// TwinCAT 3 PLC project Untitled1
// ProgramVersion: 3.1.4023.0
// libraries:
//   Tc2_ControllerToolbox, * (Beckhoff Automation GmbH)
//   Tc2_Standard, * (Beckhoff Automation GmbH)
//   Tc2_System, * (Beckhoff Automation GmbH)
//   Tc3_EventLogger, * (Beckhoff Automation GmbH)
//   Tc3_Module, * (Beckhoff Automation GmbH)
//   VisuDialogs, * (System)
//   VisuSymbols,3.5.10.0,System
// project tree:
//   DUTs/ AlarmState.TcDUT
//   / GlobalTextList.TcGTLO, PlcTask.TcTTO, Visualization Manager.TcVMO (not stored)
//   GVLs/ gAL.TcGVL
//   POUs/ ControlSystem.TcPOU, FB_EmergencySystem.TcPOU, FB_defaultValues.TcPOU, MAIN.TcPOU, FB_Tank1HysteresisBuffer.TcPOU
// real-time tasks:
//   TASK PlcTask: cycle T#10ms, priority 20, ADS port 350
// I/O:
//   DEVICE Device 1 (EtherCAT), AmsNetId 5.112.67.239.2.1
//     Term 7 (EK1200) [EK1200-5000 EtherCAT Power supply (2A E-Bus)]
//       Term 2 (EL4004) [EL4004 4Ch. Ana. Output 0-10V, 12bit]
//       Term 3 (EL4004) [EL4004 4Ch. Ana. Output 0-10V, 12bit]
//       Term 8 (EL3024) [EL3024 4Ch. Ana. Input 4-20mA DIFF]
//       Term 9 (EL3024) [EL3024 4Ch. Ana. Input 4-20mA DIFF]
//       Term 12 (EL1859) [EL1859 8Ch. Dig. Input 24V, 3ms, 8Ch. Dig. Output 24V, 0.5A]
//       Term 13 (EL9011) [EL9011 End Terminal]
// variable links:
//   Untitled1/Untitled1 Instance <-> Device 1 (EtherCAT)/Term 7 (EK1200)/Term 12 (EL1859)
//     PlcTask Inputs/MAIN.EMERGENCY_STOP <-> Channel 1/EMERGENCY STOP
//     PlcTask Inputs/MAIN.Reset_Button <-> Channel 3/Reset Button
//     PlcTask Inputs/MAIN.Toggle_Button <-> Channel 2/Toggle Button
//     PlcTask Outputs/MAIN.Motor_Direction <-> Channel 10/Motor Direction
//     PlcTask Outputs/MAIN.Motor_ON_OFF <-> Channel 9/Motor ON/OFF
//   Untitled1/Untitled1 Instance <-> Device 1 (EtherCAT)/Term 7 (EK1200)/Term 2 (EL4004)
//     PlcTask Outputs/MAIN.Flow_Valve_1 <-> AO Outputs Channel 4/Flow_Valve_1
//     PlcTask Outputs/MAIN.Level_Valve_1 <-> AO Outputs Channel 1/Level_Valve_1
//     PlcTask Outputs/MAIN.Level_Valve_2 <-> AO Outputs Channel 2/Level_Valve_2
//     PlcTask Outputs/MAIN.Level_Valve_3 <-> AO Outputs Channel 3/Level_Valve_3
//   Untitled1/Untitled1 Instance <-> Device 1 (EtherCAT)/Term 7 (EK1200)/Term 3 (EL4004)
//     PlcTask Outputs/MAIN.Gas_Valve <-> AO Outputs Channel 1/Gas_Valve
//     PlcTask Outputs/MAIN.Mixer_Valve <-> AO Outputs Channel 2/Mixer_Valve
//     PlcTask Outputs/MAIN.Motor_speed <-> AO Outputs Channel 3/Motor_Speed
//   Untitled1/Untitled1 Instance <-> Device 1 (EtherCAT)/Term 7 (EK1200)/Term 8 (EL3024)
//     PlcTask Inputs/MAIN.Pressure_Differencial_Transmitter_1 <-> AI Standard Channel 1/PDT 1
//     PlcTask Inputs/MAIN.Pressure_Differencial_Transmitter_2 <-> AI Standard Channel 3/PDT 2
//     PlcTask Inputs/MAIN.Pressure_Transmitter_1 <-> AI Standard Channel 2/PT 1
//     PlcTask Inputs/MAIN.Pressure_Transmitter_3 <-> AI Standard Channel 4/PT 3
//   Untitled1/Untitled1 Instance <-> Device 1 (EtherCAT)/Term 7 (EK1200)/Term 9 (EL3024)
//     PlcTask Inputs/MAIN.Level_Transmitter_1 <-> AI Standard Channel 2/ Level Transmitter 1
//     PlcTask Inputs/MAIN.Level_Transmitter_2 <-> AI Standard Channel 3/Level Transmitter 2
//     PlcTask Inputs/MAIN.Pressure_Transmitter_2 <-> AI Standard Channel 1/PT 2
//     PlcTask Inputs/MAIN.Temperature_Transmitter <-> AI Standard Channel 4/Temperature Transmitter

CONFIGURATION Untitled1
    RESOURCE PLC ON TwinCAT3
        TASK PlcTask(INTERVAL := T#10ms, PRIORITY := 20);
        PROGRAM MAIN WITH PlcTask : MAIN;
        PROGRAM ControlSystem WITH PlcTask : ControlSystem;
        PROGRAM BufferTankFiller WITH PlcTask : BufferTankFiller;
    END_RESOURCE
END_CONFIGURATION

// ---- DUTs/AlarmState.TcDUT
{attribute 'qualified_only'}
{attribute 'strict'}
TYPE AlarmState :
	(
		AlarmActive := 0,
		AlarmClearPreTimer := 1,
		AlarmCleared := 2
	)USINT;
END_TYPE

// ---- GVLs/gAL.TcGVL
{attribute 'qualified_only'}
VAR_GLOBAL
	fbAlarm : FB_TcAlarm;	// Creates instance of integrated Alarm FB
	
	Motor_ON_OFF 	AT %Q* : BOOL := FALSE;	// Motor switch	
	// User Input as percentage, Declaration
	Flow_Valve_1_Percentage	: INT;	// Start values
	Level_Valve_1_Percentage: INT;	// From Manual
	Level_Valve_2_Percentage: INT;
	Level_Valve_3_Percentage: INT;
	Motor_speed_Percentage	: INT; // Start speed, ideal: 30-35%
END_VAR

// ---- POUs/MAIN.TcPOU
PROGRAM MAIN
VAR
	// ------ Linking variables to IO cards ------
		// --------- Outputs ---------
	Flow_Valve_1 	AT %Q* : INT;
	Level_Valve_1 	AT %Q* : INT;
	Level_Valve_2 	AT %Q* : INT;
	Level_Valve_3 	AT %Q* : INT;
	Gas_Valve 		AT %Q* : INT;
	Mixer_Valve 	AT %Q* : INT;
	Motor_speed 	AT %Q* : INT;	
	Motor_Direction AT %Q* : BOOL; 			// Don't touch
		// --------- Inputs ---------
			// Buttons
	Toggle_Button 	AT %I* :BOOL;	// Normally Open  (OFF), Green
	Reset_Button 	AT %I* : BOOL; 	// Normally Closed (ON), Red
	EMERGENCY_STOP 	AT %I* : BOOL; 	// Normally Closed (ON), Emergency Switch
			// Sensors
	Level_Transmitter_1 	AT %I* :INT;
	Level_Transmitter_2 	AT %I* :INT;
	Temperature_Transmitter AT %I* :INT;
	Pressure_Differencial_Transmitter_1 AT %I* : INT;
	Pressure_Differencial_Transmitter_2 AT %I* : INT;
	Pressure_Transmitter_1 AT %I* : INT ;
	Pressure_Transmitter_2 AT %I* : INT ;
	Pressure_Transmitter_3 AT %I* : INT ; 
	// ------ Linking variables to IO cards ------
	
	// ------- Display Input Variables ---------
		// Percentages
	LT1percent  : INT;
	LT2percent  : INT;
	TT1percent  : INT;
	PDT1percent : INT;
	PDT2percent : INT;
	PT1percent  : INT;
	PT2percent  : INT;
	PT3percent  : INT;
		// Actual values
	LT1mm 	: REAL;
	LT2mm 	: REAL;
	TT1c 	: REAL;
	PDT1bar : REAL;
	PDT2bar : REAL;
	PT1bar  : REAL;
	PT2bar  : REAL;
	PT3bar  : REAL;
		// Scaling variables
	bitMax 		: REAL := 32767;			// [bits]
	minPT 		: REAL := 0.06;				// [bar]
	maxPT 		: REAL := 6;				// [bar]
	deltaPT 	: REAL := maxPT - minPT;	// [bar]
	minPDT		: REAL := 0.004;			// [bar]
	maxPDT		: REAL := 0.4;				// [bar]
	deltaPDT	: REAL := maxPDT - minPDT;	// [bar]
	
	//maxLT 		: REAL := 304.8;			// [mm]
	minLT1  	: REAL := 37.0;				// [mm]
	minLT1bit  	: REAL := 270.0;			// [mm]
	minLT2  	: REAL := 42.0;				// [mm]
	kLT1		: REAL := 9.0/1694.0;		// [deltaMMmeasured/deltaBitmeasured]
	kLT2		: REAL := 9.0/1529.0;		// [deltaMMmeasured/deltaBitmeasured
	
	maxTT		: REAL := 250;				// [celsius]
	minTT		: REAL := -50;				// [celsius]
	deltaTT 	: REAL := maxTT - minTT;	// [celsius]
	// ------- Display Input Variables --------- 
	
	
		// Toggle Motor Statee with green button
	risingEdge : R_TRIG;
	elapsedDebounce : TIME;
	toggleMotor : BOOL;
	
	// ------------------ HMI ------------------
	Motor_ON : BOOL; 				// For HMI button
	ON_OFF 	 : STRING(10) := 'OFF'; // For HMI text
	// ------------------ HMI ------------------
	
	// Emergency System
	alarmSystem : FB_EmergencySystem;
	
	// Initializer
	init : BOOL := FALSE;
	mainInitializer : FB_defaultValues;
END_VAR

VAR_INPUT

	Motor_ON_OFF 	AT %Q* : BOOL := FALSE;	// Motor switch	
	StartProcess : BOOL; //POU Variable for detecting machine state
	StartBuffer : BOOL := FALSE;
	
	// User Input as percentage, Declaration
	Flow_Valve_1_Percentage	: INT;
	Level_Valve_1_Percentage: INT;
	Level_Valve_2_Percentage: INT;
	Level_Valve_3_Percentage: INT;
	Motor_speed_Percentage	: INT;
END_VAR


// ======================== Initializer ========================
	IF NOT init THEN
	// ------------ Main values ------------
		mainInitializer(MotorState  := Motor_ON_OFF,
						MotorSpeed  := Motor_speed_Percentage,
						FV1_Percent := Flow_Valve_1_Percentage,
						LV1_Percent := Level_Valve_1_Percentage,
						LV2_Percent := Level_Valve_2_Percentage,
						LV3_Percent := Level_Valve_3_Percentage);
		
		init := TRUE;
	END_IF
// ======================== Initializer ========================

// ======================== Alarm System ========================
	alarmSystem(ClearButton := Reset_Button,
				EmergencyButton := EMERGENCY_STOP);
// ======================== Alarm System ========================
	
// ================ Outer bounds logic (outputs) ================
IF Flow_Valve_1_Percentage > 100 THEN
	Flow_Valve_1_Percentage := 100; 
	ELSE IF Flow_Valve_1_Percentage < 0 THEN 
		Flow_Valve_1_Percentage := 0; 
	END_IF
END_IF

IF Level_Valve_1_Percentage > 100 THEN
	Level_Valve_1_Percentage := 100; 
	ELSE IF Level_Valve_1_Percentage < 0 THEN 
		Level_Valve_1_Percentage := 0; 
	END_IF
END_IF

IF Level_Valve_2_Percentage > 100 THEN
	Level_Valve_2_Percentage := 100; 
	ELSE IF Level_Valve_2_Percentage < 0 THEN 
		Level_Valve_2_Percentage := 0; 
	END_IF
END_IF

IF Level_Valve_3_Percentage > 100 THEN
	Level_Valve_3_Percentage := 100; 
	ELSE IF Level_Valve_3_Percentage < 0 THEN 
		Level_Valve_3_Percentage := 0; 
	END_IF
END_IF

IF Motor_speed_Percentage > 100 THEN
	Motor_speed_Percentage := 100; 
	ELSE IF Motor_speed_Percentage < 0 THEN 
		Motor_speed_Percentage := 0; 
	END_IF
END_IF
// ================= Outer bounds logic (outputs) ================

// ================= Percentage Mapping (OUTPUTS) =================
	// Take 2 [V] to 10 [V]
// Flow_Valve_1 calibration
Flow_Valve_1 := REAL_TO_INT (262.14*Flow_Valve_1_Percentage +6553 ); 
// Level_Valve_1 calibration
Level_Valve_1 := REAL_TO_INT(262.14*Level_Valve_1_Percentage +6553);
// Level_Valve_2 calibration
Level_Valve_2 := REAL_TO_INT(262.14*Level_Valve_2_Percentage +6553);
// Level_Valve_3 calibration
Level_Valve_3 := REAL_TO_INT(262.14*Level_Valve_3_Percentage +6553);

// Motor_speed calibration
Motor_speed := REAL_TO_INT(262.14*Motor_speed_Percentage +6553);
// ================= Percentage Mapping (OUTPUTS) =================

// ================= Mapping (INPUTS) =================
		// Take 4 [mA] to 20 [mA] 
	// Percentages
	LT1percent  := Level_Transmitter_1;
	LT2percent  := Level_Transmitter_2;
	TT1percent  := Temperature_Transmitter;
	PDT1percent := Pressure_Differencial_Transmitter_1;
	PDT2percent := Pressure_Differencial_Transmitter_2;
	PT1percent  := Pressure_Transmitter_1;
	PT2percent  := Pressure_Transmitter_2;
	PT3percent  := Pressure_Transmitter_3;
		// Actual values
	LT1mm 	:= Level_Transmitter_1					* kLT1 						+ minLT1; // Different Mapping
	LT2mm 	:= Level_Transmitter_2 					* kLT2						+ minLT2; // Different Mapping
	TT1c 	:= Temperature_Transmitter 				* (deltaTT/bitMax)  		+ minTT;
	PDT1bar := Pressure_Differencial_Transmitter_1 	* (deltaPDT/bitMax) 		+ minPDT;
	PDT2bar := Pressure_Differencial_Transmitter_2 	* (deltaPDT/bitMax) 		+ minPDT;
	PT1bar  := Pressure_Transmitter_1 				* (deltaPT/bitMax)  		+ minPT;
	PT2bar  := Pressure_Transmitter_2 				* (deltaPT/bitMax)  		+ minPT;
	PT3bar  := Pressure_Transmitter_3 				* (deltaPT/bitMax)  		+ minPT;

	(*IF (LT1mm < 40.0) THEN
		LT1mm := 0.0;
	END_IF
	IF (LT2mm < 0.0) THEN
		LT2mm := 0.0;
	END_IF*)
// ================= Mapping (INPUTS) =================

	// Toggle motor state with green button
risingEdge(CLK := Toggle_Button,
		   Q => toggleMotor);
IF toggleMotor THEN
	Motor_ON_OFF := NOT Motor_ON_OFF;
END_IF

// ======================== HMI Display ========================
 // Start motor?
IF Motor_ON_OFF   THEN
    Motor_ON   :=  FALSE;		// Button display
	ON_OFF  := 'MOTOR: ON' ;	// Text display
	
ELSE
    Motor_ON  := TRUE;			// Button display
	ON_OFF  := 'MOTOR: OFF' ;	// Text display
END_IF
// ======================== HMI Display ========================

END_PROGRAM

// ---- POUs/FB_EmergencySystem.TcPOU
FUNCTION_BLOCK FB_EmergencySystem

VAR_INPUT			// Input variables
	ClearButton : BOOL;
	EmergencyButton : BOOL;
END_VAR

VAR					// Internal (instance) variables
	bIsInitialized : BOOL := FALSE;
	latch : BOOL := FALSE;
END_VAR

// ------------------------- Alarm Displaying ------------------------------------
IF (NOT bIsInitialized) THEN	// Initialization, since functions can't run in top pane
	bIsInitialized := TRUE;
	gAL.fbAlarm.CreateEx(TC_Events.TankAlarmEvent.Emergency, TRUE, 0);
END_IF

IF ( (NOT EmergencyButton) AND (NOT latch) ) THEN
	gAL.fbAlarm.Raise(0); // 0 -> Current time
	latch := TRUE;
END_IF

IF (EmergencyButton AND (NOT ClearButton) AND gAL.fbAlarm.bRaised) THEN
	gAL.fbAlarm.Clear(0, TRUE);	// .Clear(CurrentTime, ConfirmAlarm)
	latch := FALSE;
END_IF
// ------------------------- Alarm Displaying ------------------------------------

// ------------------------- Emergency Control -----------------------------------

// ------------------------- Emergency Control -----------------------------------

END_FUNCTION_BLOCK

// ---- POUs/FB_defaultValues.TcPOU
FUNCTION_BLOCK FB_defaultValues

VAR_IN_OUT			// Pass by Reference
	MotorState  : BOOL;
	MotorSpeed  : INT;
	FV1_Percent : INT;
	LV1_Percent : INT;
	LV2_Percent : INT;
	LV3_Percent : INT;
END_VAR

	// Definition
MotorState  := FALSE;
MotorSpeed  := 20;		 // Start speed
FV1_Percent := 100;
LV1_Percent := 100;
LV2_Percent := 100;
LV3_Percent := 0;

END_FUNCTION_BLOCK

// ---- POUs/ControlSystem.TcPOU
PROGRAM ControlSystem
VAR
		// Variables
	emergencyTime   : TIME := T#9S;
	resetLatch 		: BOOL := FALSE;
	stateAlarm 		: AlarmState := AlarmState.AlarmCleared;
	alarmTime 		: REAL;
	timeBuffer 		: TIME := T#5S;
	
		// Function Blocks
	initializer : FB_defaultValues;
	hysteresisBuffer : FB_Tank1HysteresisBuffer;
	
	// ------------------- PID -------------------
	fsetpointValue : LREAL; 	//PID setpoint
		// PID instantiation
	FB_PID : FB_CTRL_PID;					// Function Block
	ST_PIDparameters : ST_CTRL_PID_PARAMS;	// Structure
	eMode: E_CTRL_MODE;						// PID mode
		// PID Function Block Inputs
	setPoint : LREAL;
	fActualValue   : LREAL;
	fManSyncValue  : LREAL;
	bSync          : BOOL;
	bHold          : BOOL;
	fOutBuffer 	   : LREAL;
	// ------------------- PID -------------------
END_VAR

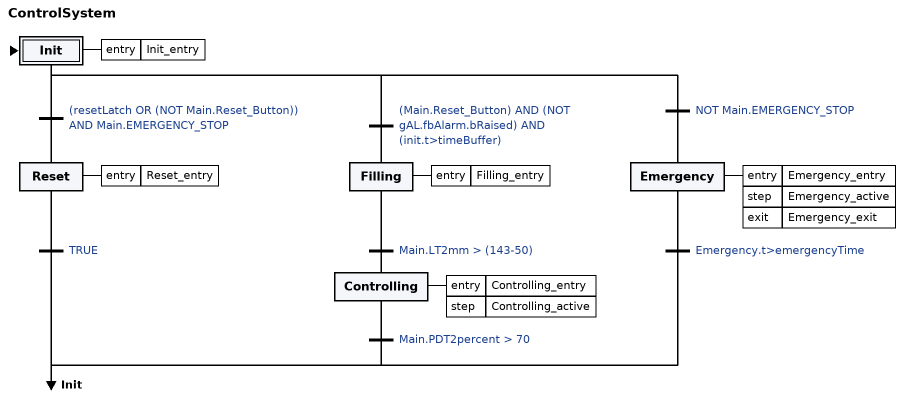
INITIAL_STEP Init:
    Init_entry(P1);  // entry action
END_STEP
TRANSITION FROM Init TO Reset
    := (resetLatch OR (NOT Main.Reset_Button)) AND Main.EMERGENCY_STOP;
END_TRANSITION
STEP Reset:
    Reset_entry(P1);  // entry action
END_STEP
TRANSITION FROM Reset TO Init
    := TRUE;
END_TRANSITION
TRANSITION FROM Init TO Filling
    := (Main.Reset_Button) AND (NOT gAL.fbAlarm.bRaised) AND (init.t>timeBuffer);
END_TRANSITION
STEP Filling:
    Filling_entry(P1);  // entry action
END_STEP
TRANSITION FROM Filling TO Controlling
    := Main.LT2mm > (143-50);
END_TRANSITION
STEP Controlling:
    Controlling_entry(P1);  // entry action
    Controlling_active(N);  // step action
END_STEP
TRANSITION FROM Controlling TO Init
    := Main.PDT2percent > 70;
END_TRANSITION
TRANSITION FROM Init TO Emergency
    := NOT Main.EMERGENCY_STOP;
END_TRANSITION
STEP Emergency:
    Emergency_entry(P1);  // entry action
    Emergency_active(N);  // step action
    Emergency_exit(P0);  // exit action
END_STEP
TRANSITION FROM Emergency TO Init
    := Emergency.t>emergencyTime;
END_TRANSITION

ACTION Controlling_active:

// ========== Buffer Hysteresis for Tank 1 ===========
	hysteresisBuffer(motorOnOff => Main.Motor_ON_OFF);
// ========== Buffer Hysteresis for Tank 1 ===========

(*
// =========== Control Algoritm with PID =============
	FB_PID( fSetpointValue 	:= 	setPoint,		// Desired Value
			fActualValue 	:= 	Main.LT2mm,		// Actual  Value
			fManSyncValue 	:= 	fManSyncValue,
			bSync 			:= 	bSync,
			eMode 			:= 	eMode,			// PID mode - manual
			bHold 			:= 	bHold,				// Hold output at current value
			stParams 		:= 	ST_PIDparameters,
			fOut 			=> 	fOutBuffer );
	// PID FB also takes in the struct values, not specified here.
	Main.Level_Valve_1_Percentage := LREAL_TO_INT(fOutBuffer);
// =========== Control Algoritm with PID =============
*)
END_ACTION

ACTION Controlling_entry:
	// Controlling initialization
Main.Level_Valve_1_Percentage := 45;
Main.Level_Valve_2_Percentage := 100;	// Open
Main.Level_Valve_3_Percentage := 0;		// Closed
END_ACTION

ACTION Emergency_active:

IF ( (Main.EMERGENCY_STOP) AND (NOT Main.Reset_Button) ) THEN
	resetLatch := TRUE;
	stateAlarm := AlarmState.AlarmClearPreTimer;
END_IF

IF resetLatch THEN
	alarmTime := TIME_TO_REAL(emergencyTime - emergency.t)/1000;
END_IF
END_ACTION

ACTION Emergency_entry:

Main.Motor_ON_OFF := FALSE;				// Stop Motor
Main.Flow_Valve_1_Percentage  := 100;	// Open all valves
Main.Level_Valve_1_Percentage := 100;
Main.Level_Valve_2_Percentage := 100;
Main.Level_Valve_3_Percentage := 100;

stateAlarm := AlarmState.AlarmActive;
END_ACTION

ACTION Emergency_exit:

alarmTime := 0.0;
END_ACTION

ACTION Filling_entry:
	// Start Filling
Main.Motor_ON_OFF := TRUE;				// ON
Main.Flow_Valve_1_Percentage  := 100;	// Open
Main.Level_Valve_1_Percentage := 100;	// Open
Main.Level_Valve_2_Percentage := 0;		// Closed
Main.Level_Valve_3_Percentage := 100;	// Open
END_ACTION

ACTION Init_entry:

// ------------ Initialize PID Values ------------
	ST_PIDparameters.tTaskCycleTime := T#10MS;	// Cycle Time, PLC
	ST_PIDparameters.tCtrlCycleTime := T#10MS;	// Cycle Time, Controller
	ST_PIDparameters.fOutMaxLimit 	:= 100; 	// Max allowed output - 100% valve
	ST_PIDparameters.fOutMinLimit 	:= 15; 		// Min allowed output - LV2 closed with deadzone
	eMode := eCTRL_MODE_Manual; 				// Set PID control mode to manual
	
	ST_PIDparameters.fKp 			:= 0.00001;	// K_P ~ Proportional Gain
	ST_PIDparameters.tTn 			:= T#1MS;	// K_I ~ Integral Time Constant
	ST_PIDparameters.tTv 			:= T#1MS;	// K_D ~ Derivative Time Constant
	ST_PIDparameters.tTd 			:= T#10MS;	// Filter time for derivative
	
	fSetpointValue := 140;
END_ACTION

ACTION Reset_entry:

initializer(MotorState  := Main.Motor_ON_OFF,
			MotorSpeed  := Main.Motor_speed_Percentage,
			FV1_Percent := Main.Flow_Valve_1_Percentage,
			LV1_Percent := Main.Level_Valve_1_Percentage,
			LV2_Percent := Main.Level_Valve_2_Percentage,
			LV3_Percent := Main.Level_Valve_3_Percentage);

stateAlarm := AlarmState.AlarmCleared;
resetLatch := FALSE;
END_ACTION

END_PROGRAM

// ---- POUs/FB_Tank1HysteresisBuffer.TcPOU
FUNCTION_BLOCK FB_Tank1HysteresisBuffer

VAR_OUTPUT
	motorOnOff : BOOL;
END_VAR

VAR
	minLT1mm : REAL := 50.0;
	maxLT1mm : REAL := 60.0;
END_VAR

	// To keep water in tank 1
IF main.LT1mm > maxLT1mm THEN
	motorOnOff := FALSE;
ELSIF main.LT1mm < minLT1mm THEN
	motorOnOff := TRUE; 
END_IF

END_FUNCTION_BLOCK

// ---- GlobalTextList.TcGTLO
TEXTLIST GlobalTextList
  9 = '%f'
  594 = '%I'
  907 = '%i'
  617 = 'aaaaaaaa'
  411 = 'EMERGENCY STOP'
  749 = 'EMERGENCY STOP %s'
  283 = 'Flow Valve %i'
  422 = 'Flow Valve 1 = %f %'
  201 = 'Flow Valve = %i'
  842 = 'Flow Valve: %i'
  336 = 'Flow Valve: %i %'
  590 = 'Flow Valve: %i%'
  567 = 'Gas Valve : %i%'
  736 = 'Level Valve 1 = %f %'
  833 = 'Level Valve 1 = %i %'
  36 = 'Level Valve 1: %i'
  942 = 'Level Valve 1: %i%'
  802 = 'Level Valve 2: %i%'
  940 = 'Level Valve 3: %i%'
  781 = 'Mixer Valve : %i%'
  1 = 'Motor   %s'
  109 = 'Motor Direction %s'
  202 = 'Motor OFF'
  60 = 'Motor OFF  '
  480 = 'Motor OFF  %B'
  834 = 'Motor OFF  %s'
  840 = 'Motor ON'
  885 = 'MOtor ON'
  981 = 'Motor Speed: %i%'
  390 = 'PDT 1'
  74 = 'PDT 1 %i'
  240 = 'PDT 1 = %.4f  Bar'
  2 = 'PDT 1 = %4.f  Bar'
  419 = 'PDT 1 = %4f  Bar'
  414 = 'PDT 1 = %f Bar'
  882 = 'PDT 1 = %f.4 Bar'
  541 = 'PDT 1 = %fmaxDecimals = 3 Bar'
  384 = 'PDT 1 = %i'
  145 = 'PDT 1 = %i Bar'
  423 = 'PDT 2 %i'
  214 = 'PDT 2 = %.4f Bar'
  437 = 'PDT 2 = %f Bar'
  723 = 'PDT 2 = %i'
  493 = 'PDT 2 = %i Bar'
  589 = 'PT 1 %i'
  999 = 'PT 1 = %.4f Bar'
  314 = 'PT 1 = %f Bar'
  203 = 'PT 1 = %i Bar'
  730 = 'sdfsdf'
  313 = 'START'
  187 = 'START %s'
  945 = 'STOP'
  921 = 'STOP %s'
END_TEXTLIST
